FUNCTION_BLOCK AB_KOSCMD_RECEIVER (* Simple FB with one algorithm *)
  (* Standard: 61499-1 *)
  (* Version 1.0, 2023-05-24, test *)
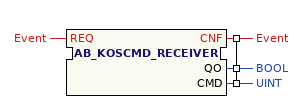
  EVENT_INPUT
    REQ; (* Normal Execution Request *)
  END_EVENT
  EVENT_OUTPUT
    CNF WITH CMD, QO; (* Execution Confirmation *)
  END_EVENT
  VAR_OUTPUT
    QO : BOOL;
    CMD : UINT;
  END_VAR
  ALGORITHM REQ IN ST:

  END_ALGORITHM
END_FUNCTION_BLOCK
